TYPE st_SafetyByPass :
STRUCT
	SafeDoorByPass :BOOL := FALSE;
	//AliveCheckingBYPass : BOOL;
END_STRUCT
END_TYPE

(* stored: Version 1.1.0.1, ProductVersion 3.1.4024.13
   DUT st_SafetyByPass: Id {a9b9684b-8783-4786-9450-01b4f7850c88} *)
